// SIMATIC STEP 7 (V5.x) project FILLING
// program: S7 Program(1)

SYMBOL_TABLE
"FILLING_CYCLE"	FB 145	FB 145	// Цикл наполнения илоуплотнителей
END_SYMBOL_TABLE

FUNCTION_BLOCK "FILLING_CYCLE"	// FB 145
TITLE = Циклическая работа затвора 13 на уплотнителях ила
//Уровень ила в резервуарах не учитывается, так как стоят стоят датчики мутности 
//вместо датчиков уровня ила. 
//Блок управляет только общим затвором №13. Для управления затвором используется 
//ранее написанный драйвер в ПЛК1_1. Минимальный шаг времени - 10 секунд.
//
//Ручной режим управления задается в блоке затвора, в данном блоке MAN 
//обрабатывает возможные аварии и может формировать сигнал ПАЗ. Так же если 
//включен ручной режим, через MAN идет пропуск выполнения данного блока.
//
//В SCADA необходимо будет сделать обратный счет времени, тогда как тут идет 
//прямой счет.
//
//В данном блоке используется следующая переферия:
//Таймеры:  T0, T1, T5
//Счетчики: C0, C1
//
//Для затворов слива (цикла слива илоуплотнителей) ила используется отдельный 
//блок.
AUTHOR : ETSystem
VERSION : 0.1
VAR_INPUT
  OPENED : BOOL ;	//Затвор открыт
  CLOSED : BOOL ;	//Затвор закрыт
  G_FAULT : BOOL ;	//Ошибка на затворе
  C_FAULT : BOOL ;	//Ошибка коммуникации
  AUTO_ON : BOOL ;	//Автоматический режим включен
  CLOSE_IF_STOP : BOOL ;	//Закрывать затвор если нажата кнопка СТОП
  WT_TASK : INT  := 3;	//Время работы (задание)
  DT_TASK : INT  := 5;	//Время простоя (задание)
  T_BASE : S5TIME  := S5T#5S;	//База времени поделенная на 2 (исп. 2 таймера)
END_VAR
VAR_OUTPUT
  QON_OPENING : BOOL ;	//Команда на открытие затвора
  QON_CLOSING : BOOL ;	//Команда на закрытие затвора
  QCOMMON_FAULT : BOOL ;	//Общая ошибка
  START_OS_MSG : BOOL ;	//В ПЛК - индикация нажатия кнопки, в OS - обратная связь что кнопка была нажата
  STOP_OS_MSG : BOOL ;	//В ПЛК - индикация нажатия кнопки, в OS - обратная связь что кнопка была нажата
  FILLING_MODE : BOOL ;	//Активен режим наполнения
  WAITING_MODE : BOOL ;	//Активен режим ожидания
  CYCLE_STATUS : BOOL ;	//Цикл запущен
  CNT_FILLING : INT ;	//Счетчик наливов илоуплотнителей
  QWT : INT ;	//Текущее отработанное время (в итерации цикла)
  QDT : INT ;	//Текущее время простоя (в итерации цикла)
END_VAR
VAR_IN_OUT
  START_OS : BOOL ;	//Старт цикла - со СКАДА (OS)
  STOP_OS : BOOL ;	//Стоп цикла - со СКАДА (OS)
END_VAR
VAR
  T1_RESET : BOOL ;	//Сброс таймера 1
  C1_RESET : BOOL ;	//Сброс счетчика 1
  COMMON_FAULT : BOOL ;	//Общая ошибка блока
  FIRST_TIME_AUTO : BOOL  := TRUE;	//Автоматический режим запущен в первый раз (1 - да, 0 - нет)
  WT_FLAG : BOOL ;	//Флаг режима налива (1), слива (0)
  FP_START : BOOL ;	//Нарастающий фронт кнопки START
  FP_STOP : BOOL ;	//Нарастающий фронт кнопки STOP
  AUTO_STATUS : BOOL ;	//Автоматический режим был включен
  FP_TICK : BOOL ;
END_VAR
BEGIN
NETWORK
TITLE = Определение наличия аварий или нештатных ситуаций.
//Для определения режима работы используем внешнюю переменную DB10.ZV13_Auto с 
//PLC1_1: 0 - дист., 1 - авто, если автоматический режим не включен, переходим к 
//выходу из автоматического режима (в MAN).
//В качестве общей аварии используем только аварии которые определяет данный 
//блок.
//!!! Проверяем включен ли вообще автоматический режим если нет уходим из блока
      AN    #AUTO_ON;
      JC    MAN;
      A     #AUTO_STATUS;
      JC    AUTO;
//Проверяем корректность запуска автоматического режима (если затвор не закрыт)
//То запуск невозможен, надо выдать ошибку на блок ПАЗ затвора и выйти из автомата
      AN    #CLOSED;
      S     #COMMON_FAULT;
      JC    MAN;
//Или устанавливаем параметр запуска автоматического режима AUTO_STATUS:
      A     #CLOSED;
      S     #AUTO_STATUS;
AUTO: NOP   0;
//!!! Возможные ошибки, если есть уходим из блока
//Внешние сигналы с блока управления затвором
//Авария на затворе ИЛИ Авария по связи 
      O     #G_FAULT;
      JC    MAN;
      O     #C_FAULT;
//Установим флаг общей аварии и перейдем к обработчику
      =     #COMMON_FAULT;
//Если есть какая-то авария, переинициализируем автоматический режим
      JC    MAN;
//Данный сигнал будет заведен в ПАЗ, которая идолжна будет отработать закрытие клапана
//и перевод его в режим ручной работы. Настройки PAZ блока управления затвором:
//EN_PAZ = ВКЛ, OFF_PAZ1 = Закрывать при аварии, PAZ_GONE = Оставлять в состоянии ПАЗ
//PAZ_MODE = Включать ручной режим
//Кроме того сбрасываем сигналы на открытие/закрытие задвижки если она открыта/закрыта
//      A     #OPENED
//    R     #QON_OPENING
//  A     #CLOSED
//R     #QON_CLOSING
      A     #QON_OPENING;
      A     #OPENED;
      O(;
      A     #QON_OPENING;
      AN    #OPENED;
      AN    #CLOSED;
      );
      R     #QON_OPENING;
      A     #QON_CLOSING;
      A     #CLOSED;
      O(;
      A     #QON_CLOSING;
      AN    #OPENED;
      AN    #CLOSED;
      );
      R     #QON_CLOSING;
//Либо управляем импульсами:
//Открытие:
// A     #QON_OPENING
//   L     S5T#3S
//     SP    T      5
//     A     T      5
//      =     #QON_OPENING
//Закрытие:
//     A     #QON_CLOSING
//      L     S5T#3S
//      SP    T      5
//      A     T      5
//      =     #QON_CLOSING
NETWORK
TITLE = Обработка кнопок
//В данном блоке реализованы три кнопки:
//START - сбрасывает всю статистику и запускает цикл по новой (неактивна при 
//запущенном цикле).
//STOP - Останавливает выполнение цикла, сохраняет статистику (неактивна после 
//нажания), так же если настройка CLOSE_IF_STOP активирована, закрывает затвор. 
//Кнопка STOP заблокирована если затвор находится в промежуточном положении.
//Обработка кнопок, ловим передний импульс (FP) по кнопке и фиксируем его (S)
//Так же сбрасываем все остальные статусы кнопок (R) 
//Кнопка START:
      A     #START_OS;
      FP    #FP_START;
      R     #START_OS;
      S     #START_OS_MSG;
      R     #STOP_OS_MSG;
//Кнопка STOP:
      A     #STOP_OS;
      FP    #FP_STOP;
      R     #STOP_OS;
      S     #STOP_OS_MSG;
      R     #START_OS_MSG;
NETWORK
TITLE = Определение режима работы блока START/STOP
//Смотрим какая кнопка была нажата, в любом случае выставляем выход QAUTO, для 
//отладки. И как флаг того что автоматический режим был запущен без ошибок.
      A     #STOP_OS_MSG;
      JC    STOP;
      A     #START_OS_MSG;
      JCN   N1;
NETWORK
TITLE = Автоматический режим налива (в цикле)
//Автоматический режим налива на основе двух таймеров и триггера, база времени 
//заданна в размере 10 секунд (два таймера по 5 секунд).
//
//Если первое включение автоматического режима, инициализируем его
      AN    #FIRST_TIME_AUTO;
      JC    A_C;
//Если ошибок нет, сбрасываем флаг первого запуска автоматического режима,
//значения на счетчиках, таймеры, флаги сбросов, и флага налива подаем 
// команду на открытие затвора
      AN    #COMMON_FAULT;
      R     #FIRST_TIME_AUTO;
      R     C 1;
      R     C 0;
      R     T 1;
      R     T 0;
      R     #T1_RESET;
      S     #C1_RESET;
      S     #QON_OPENING;
      S     #WT_FLAG;
//Включим индикацию запуска наполнения
      S     #CYCLE_STATUS;
//Обнулим счетчики
      L     0;
      T     #QWT;
      T     #QDT;
      T     #CNT_FILLING;
//Для отсчета времени используется два таймера T1, T2 и один триггер,
//для задания верной частоты работы таймера необходимо записать в каждый таймер
//значение в два раза меньшее чем необходимое время отсчета (для 1 сек, 500мс)
//Триггер (и соответственно счет) запускается если затвор полность открыт, 
//или полность закрыт, при этом нет никаких аварий, иначе, останавливаем таймер,  
//сбрасываем счетчик, выходим из автоматического режима в ручной
A_C:  NOP   0;
//Если задвижка открывается или закрывается, то ничего не считываем
//Надо считывать открывается или закрывается у нас затвор, либо 
//проверятьчто он ИЛИ открыт, ИЛИ закрыт.
//      O     #QON_OPENING
//      O     #QON_CLOSING
      AN    #CLOSED;
      AN    #OPENED;
      JC    N1;
//Таймер 2
      AN    T 1;
      AN    #C1_RESET;
      L     #T_BASE;
      SE    T 0;
//Триггер (условие запуска)
      AN    #C1_RESET;
      A(;
      A     #OPENED;
      A     #WT_FLAG;
      O;
      A     #CLOSED;
      AN    #WT_FLAG;
      );
      S     #T1_RESET;
      A     T 0;
      R     #T1_RESET;
//Таймер 1
      A     #T1_RESET;
      L     #T_BASE;
      SE    T 1;
//Счетчик 1
      A     #C1_RESET;
      R     C 1;
      AN    T 1;
//AN    #C1_RESET
      FP    #FP_TICK;
      CU    C 1;
//Определяем какой цикл считается (для правильного сброса)
//Рабочий?
      A     #OPENED;
      A     #WT_FLAG;
      JC    WT_C;
//Простоя?
      A     #CLOSED;
      AN    #WT_FLAG;
      JC    DT_C;
//Иначе ждем открытия, либо закрытия затвора 13
      JU    N1;
//В симуляторе не устанавливается вовремя C1_RESET после операции простоя
//это нужно иметь ввиду и проверить на реальном устройстве
//Рабочий цикл
WT_C: NOP   0;
//Проверяем значение в счетчике > WT_TASK сбрасываем:
      L     C 1;
      T     #QWT;	//Выход отсчета
      L     #WT_TASK;	//Время со входа в блок в минутах
//Требуемое время истекло
      >=I;
      S     #C1_RESET;	//Сбрасываем счетчик
      S     #QON_CLOSING;	//Отправляем сигнал на закрытие
//Сменим флаг режима
      R     #WT_FLAG;
//И сбросим индикацию рабочего режима
      R     #FILLING_MODE;
//Увеличиваем счетчик циклов налива на 1
      CU    C 0;
//Или продолжаем считать
      <I;
      R     #C1_RESET;
//Устанавливаем флаг режима наполнения и сбрасываем флаг ожидания
      S     #FILLING_MODE;
      L     C 0;
      T     #CNT_FILLING;
      JU    N1;
//Цикл ожидания
DT_C: NOP   0;
//Проверяем значение в счетчике > DT_TASK сбрасываем:
      L     C 1;
      T     #QDT;
      L     #DT_TASK;	//Время со входа в блок в минутах
//Требуемое время истекло
      >=I;
      S     #C1_RESET;	//Сбрасываем счетчик
      S     #QON_OPENING;	//Отправляем сигнал на открытие
//Сменим флаг режима
      S     #WT_FLAG;
//И сбросим индикацию режима ожидания
      R     #WAITING_MODE;
//Или продолжаем считать
      <I;
      R     #C1_RESET;
//Устанавливаем флаг режима ожидания и сбрасываем флаг наполнения
      S     #WAITING_MODE;
      JU    N1;
NETWORK
TITLE = STOP MODE
//Останавливаем счет, при этом не сбрасываем статистику, если задан параметр 
//CLOSE_IF_STOP закрываем затвор. Кроме того для верной инициализации режима 
//налива сбрасываем инициализацию автоматического режима, при его повторном 
//запуске, цикл начнется с нуля. Если STOP осущетсвляется когда затвор находится 
//в 
//промежуточном положении, выходим по ошибке.
STOP: NOP   0;
      SET;
      R     #STOP_OS_MSG;
      R     T 1;
      R     T 0;
      A     #CLOSE_IF_STOP;
      AN    #CLOSED;
      S     #QON_CLOSING;
      AN    #FIRST_TIME_AUTO;
      S     #FIRST_TIME_AUTO;
//Выключим индикацию запуска наполнения
      A     #CYCLE_STATUS;
      R     #CYCLE_STATUS;
//Сбросим индикацию режимов работы
      A     #FILLING_MODE;
      R     #FILLING_MODE;
      A     #WAITING_MODE;
      R     #WAITING_MODE;
      JU    N1;
NETWORK
TITLE = Переход из авто в ручной, и обработка аварий
MAN:  NOP   0;
//Не в автоматическом режиме и не были в нем, но при этом затвор закрыт
//Сбросим ошибку на блоке если мы в ручном режиме и затвор закрыт.
      AN    #AUTO_ON;
      AN    #AUTO_STATUS;
      A     #CLOSED;
      R     #QCOMMON_FAULT;
      JC    N1;
//!!! Иначе были в автоматическом, но что-то пошло не так, тогда
//сбрасываем настройки автоматического режима:
//Если сброшен бит первого запуска автоматического режима, установим его
//для того чтобы при переходе из ручного в автоматический и наоборот
//автоматический режим верно инициализировался со сбросом счетчиков
      AN    #FIRST_TIME_AUTO;
      S     #FIRST_TIME_AUTO;
//Если автоматический режим выключен, или авария обнулим выходы счетчиков
      L     0;
      T     #QDT;
      T     #QWT;
//Счетчик цикла
      T     #CNT_FILLING;
//Сбрасываем различные условия работы автоматического режима, мы не в автомате
      SET;
      R     #START_OS_MSG;
      R     #STOP_OS_MSG;
      R     #AUTO_STATUS;
//Выключим индикацию запуска наполнения
      R     #CYCLE_STATUS;
//Сбросим индикацию режимов работы
      R     #FILLING_MODE;
      R     #WAITING_MODE;
//Заодно если идет открытие или закрытие, сбрасываем эти сигналы:
//На всякий случай так, удалить при отладке
      R     #QON_OPENING;
      R     #QON_CLOSING;
//Группируем ошибки в одну, с учетом что если автоматический режим не включен
//то нам не важно открыта заслонка или закрыта
      O     #COMMON_FAULT;
      =     #QCOMMON_FAULT;
      JU    N1;
NETWORK
TITLE = Завершаем выполнение блока
//Заменить все переходы сюда на BE, после того как код будет полностью отлажен.
N1:   NOP   0;
END_FUNCTION_BLOCK

ORGANIZATION_BLOCK OB 1
TITLE = "Main Program Sweep (Cycle)"
VERSION : 0.1
VAR_TEMP
  OB1_EV_CLASS : BYTE ;	//Bits 0-3 = 1 (Coming event), Bits 4-7 = 1 (Event class 1)
  OB1_SCAN_1 : BYTE ;	//1 (Cold restart scan 1 of OB 1), 3 (Scan 2-n of OB 1)
  OB1_PRIORITY : BYTE ;	//Priority of OB Execution
  OB1_OB_NUMBR : BYTE ;	//1 (Organization block 1, OB1)
  OB1_RESERVED_1 : BYTE ;	//Reserved for system
  OB1_RESERVED_2 : BYTE ;	//Reserved for system
  OB1_PREV_CYCLE : INT ;	//Cycle time of previous OB1 scan (milliseconds)
  OB1_MIN_CYCLE : INT ;	//Minimum cycle time of OB1 (milliseconds)
  OB1_MAX_CYCLE : INT ;	//Maximum cycle time of OB1 (milliseconds)
  OB1_DATE_TIME : DATE_AND_TIME ;	//Date and time OB1 started
END_VAR
BEGIN
// (block stored without names or comments; labels and parameter names are numbered)
END_ORGANIZATION_BLOCK
